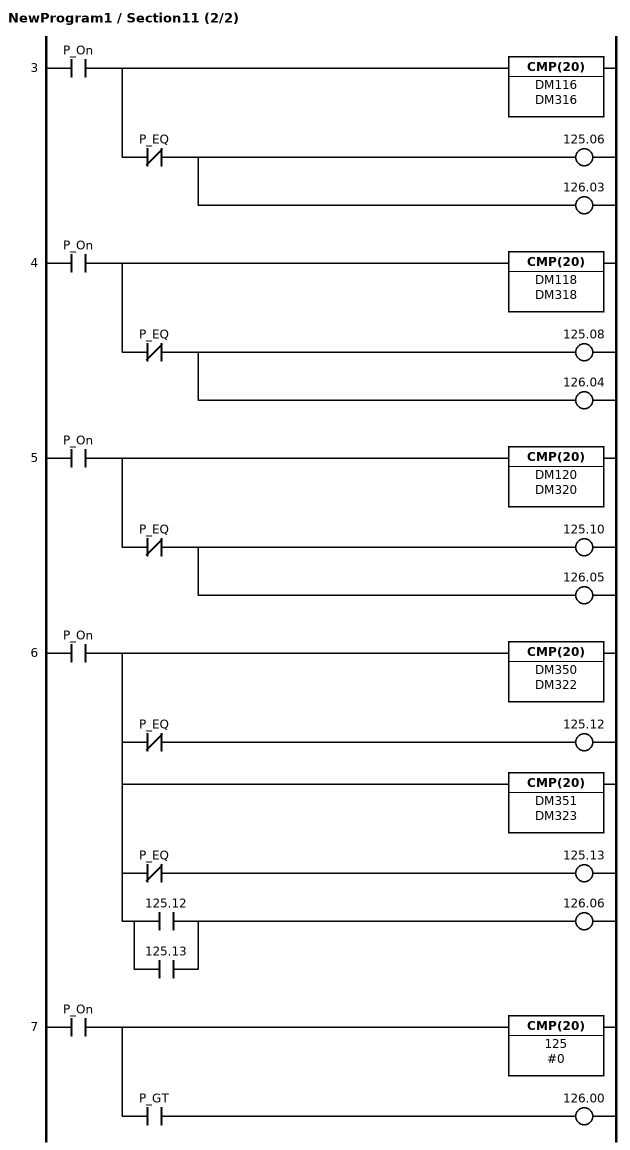
; [picture p48: NewProgram1 / Section11, rungs 3-7]
; rung 3
LD P_On
CMP(20) DM116 DM316
ANDNOT P_EQ
OUT 125.06
OUT 126.03
; rung 4
LD P_On
CMP(20) DM118 DM318
ANDNOT P_EQ
OUT 125.08
OUT 126.04
; rung 5
LD P_On
CMP(20) DM120 DM320
ANDNOT P_EQ
OUT 125.10
OUT 126.05
; rung 6
LD P_On
OUT TR0
CMP(20) DM350 DM322
ANDNOT P_EQ
OUT 125.12
LD TR0
CMP(20) DM351 DM323
ANDNOT P_EQ
OUT 125.13
LD TR0
LD 125.12
OR 125.13
ANDLD
OUT 126.06
; rung 7
LD P_On
CMP(20) 125 #0
AND P_GT
OUT 126.00

### Section Section12

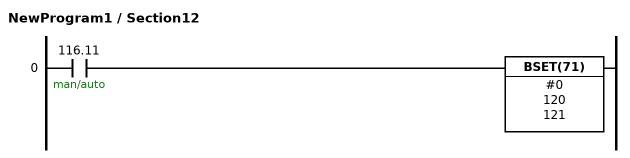
; rung 0
LD 116.11  ; man/auto
BSET(71) #0 120 121

### Section Section13

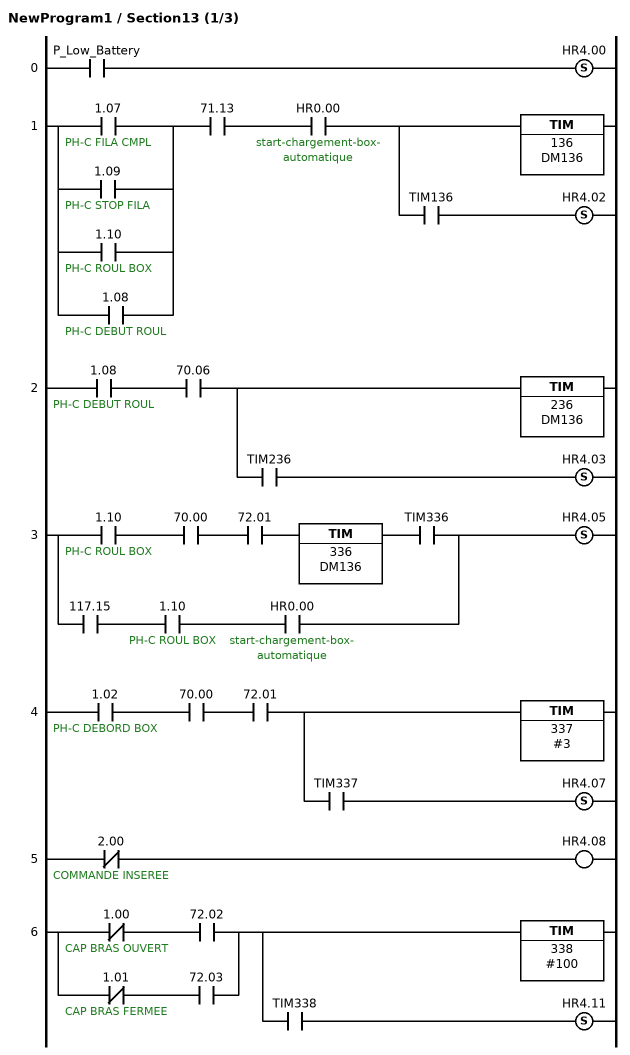
; rung 0
LD P_Low_Battery
SET HR4.00
; rung 1
LD 1.07  ; PH-C FILA CMPL
OR 1.09  ; PH-C STOP FILA
OR 1.10  ; PH-C ROUL BOX
OR 1.08  ; PH-C DEBUT ROUL
AND 71.13
AND HR0.00  ; start-chargement-box-automatique
TIM 136 DM136
AND TIM136
SET HR4.02
; rung 2
LD 1.08  ; PH-C DEBUT ROUL
AND 70.06
TIM 236 DM136
AND TIM236
SET HR4.03
; rung 3
LD 1.10  ; PH-C ROUL BOX
AND 70.00
AND 72.01
TIM 336 DM136
AND TIM336
LD 117.15
AND 1.10  ; PH-C ROUL BOX
AND HR0.00  ; start-chargement-box-automatique
ORLD
SET HR4.05
; rung 4
LD 1.02  ; PH-C DEBORD BOX
AND 70.00
AND 72.01
TIM 337 #3
AND TIM337
SET HR4.07
; rung 5
LDNOT 2.00  ; COMMANDE INSEREE
OUT HR4.08
; rung 6
LDNOT 1.00  ; CAP BRAS OUVERT
AND 72.02
LDNOT 1.01  ; CAP BRAS FERMEE
AND 72.03
ORLD
TIM 338 #100
AND TIM338
SET HR4.11

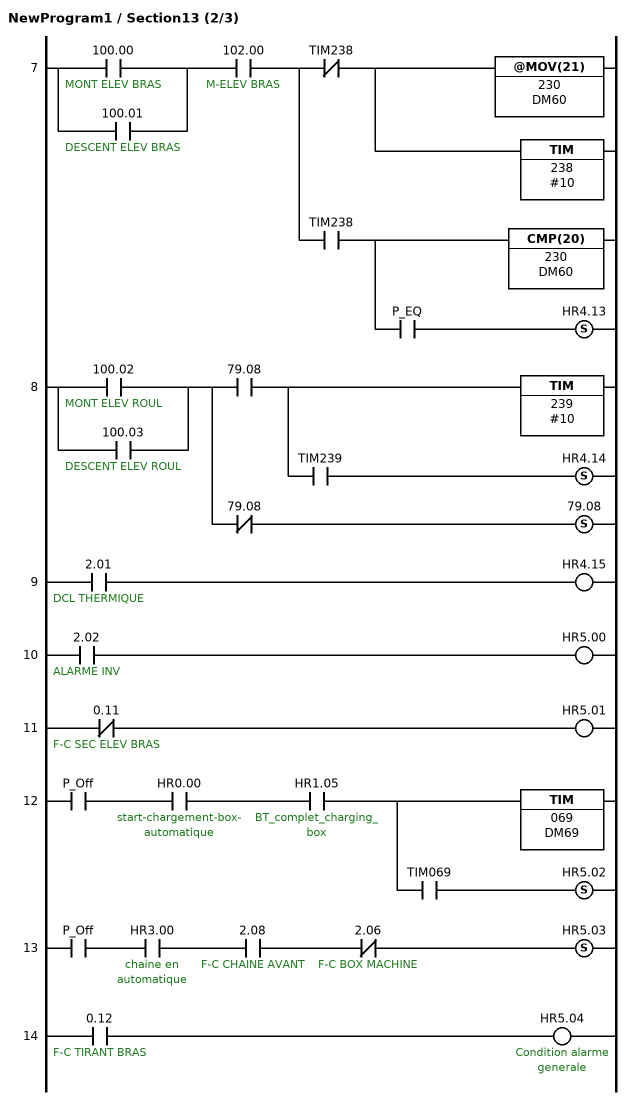
; rung 7
LD 100.00  ; MONT ELEV BRAS
OR 100.01  ; DESCENT ELEV BRAS
AND 102.00  ; M-ELEV BRAS
OUT TR0
ANDNOT TIM238
@MOV(21) 230 DM60
TIM 238 #10
LD TR0
AND TIM238
CMP(20) 230 DM60
AND P_EQ
SET HR4.13
; rung 8
LD 100.02  ; MONT ELEV ROUL
OR 100.03  ; DESCENT ELEV ROUL
OUT TR0
AND 79.08
TIM 239 #10
AND TIM239
SET HR4.14
LD TR0
ANDNOT 79.08
SET 79.08
; rung 9
LD 2.01  ; DCL THERMIQUE
OUT HR4.15
; rung 10
LD 2.02  ; ALARME INV
OUT HR5.00
; rung 11
LDNOT 0.11  ; F-C SEC ELEV BRAS
OUT HR5.01
; rung 12
LD P_Off
AND HR0.00  ; start-chargement-box-automatique
AND HR1.05  ; BT_complet_charging_box
TIM 069 DM69
AND TIM069
SET HR5.02
; rung 13
LD P_Off
AND HR3.00  ; chaine en automatique
AND 2.08  ; F-C CHAINE AVANT
ANDNOT 2.06  ; F-C BOX MACHINE
SET HR5.03
; rung 14
LD 0.12  ; F-C TIRANT BRAS
OUT HR5.04  ; Condition alarme generale

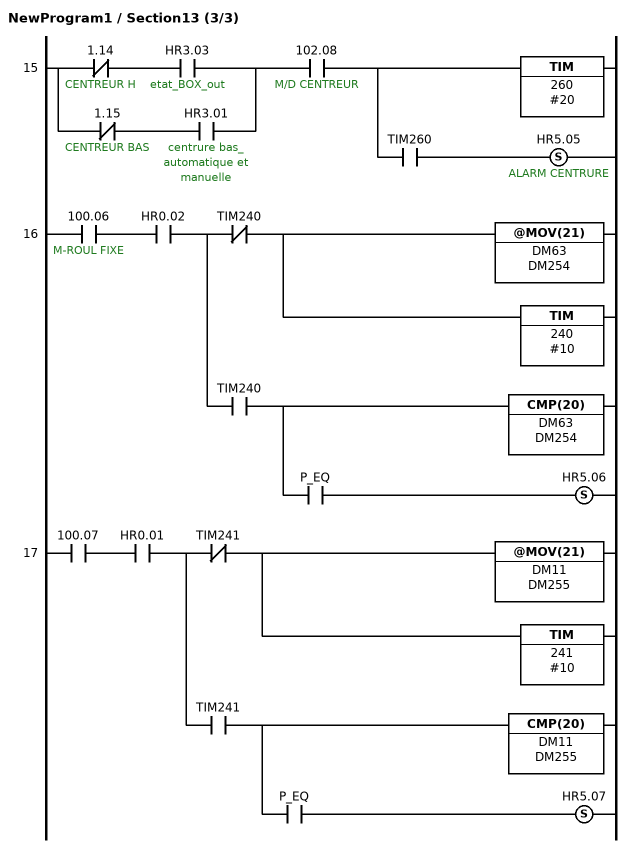
; rung 15
LDNOT 1.14  ; CENTREUR H
AND HR3.03  ; etat_BOX_out
LDNOT 1.15  ; CENTREUR BAS
AND HR3.01  ; centrure bas_automatique et manuelle
ORLD
AND 102.08  ; M/D CENTREUR
TIM 260 #20
AND TIM260
SET HR5.05  ; ALARM CENTRURE
; rung 16
LD 100.06  ; M-ROUL FIXE
AND HR0.02
OUT TR0
ANDNOT TIM240
@MOV(21) DM63 DM254
TIM 240 #10
LD TR0
AND TIM240
CMP(20) DM63 DM254
AND P_EQ
SET HR5.06
; rung 17
LD 100.07
AND HR0.01
OUT TR0
ANDNOT TIM241
@MOV(21) DM11 DM255
TIM 241 #10
LD TR0
AND TIM241
CMP(20) DM11 DM255
AND P_EQ
SET HR5.07

### Section consentement

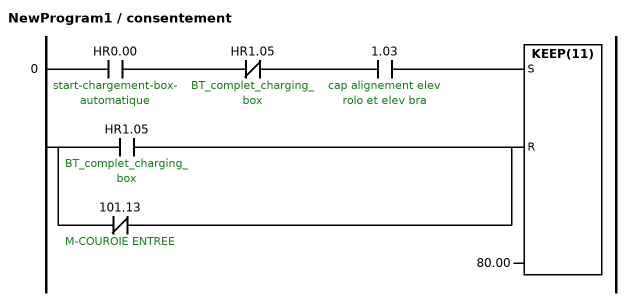
; rung 0
LD HR0.00  ; start-chargement-box-automatique
ANDNOT HR1.05  ; BT_complet_charging_box
AND 1.03  ; cap alignement elev rolo et elev bra
LD HR1.05  ; BT_complet_charging_box
ORNOT 101.13  ; M-COUROIE ENTREE
KEEP(11) 80.00

### Section Section15

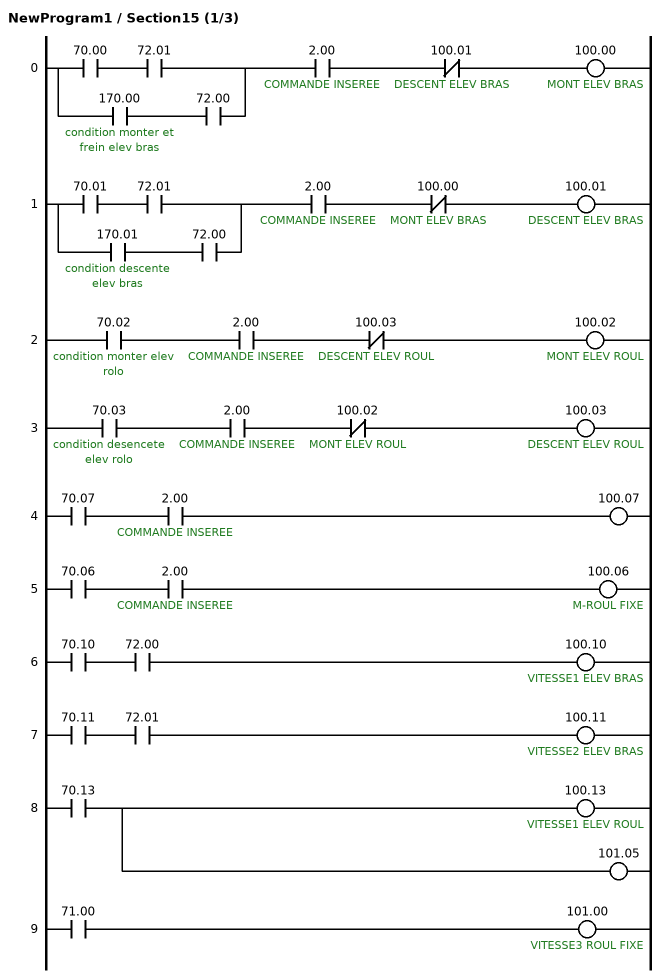
; rung 0
LD 70.00
AND 72.01
LD 170.00  ; condition monter et frein elev bras
AND 72.00
ORLD
AND 2.00  ; COMMANDE INSEREE
ANDNOT 100.01  ; DESCENT ELEV BRAS
OUT 100.00  ; MONT ELEV BRAS
; rung 1
LD 70.01
AND 72.01
LD 170.01  ; condition descente elev bras
AND 72.00
ORLD
AND 2.00  ; COMMANDE INSEREE
ANDNOT 100.00  ; MONT ELEV BRAS
OUT 100.01  ; DESCENT ELEV BRAS
; rung 2
LD 70.02  ; condition monter elev rolo
AND 2.00  ; COMMANDE INSEREE
ANDNOT 100.03  ; DESCENT ELEV ROUL
OUT 100.02  ; MONT ELEV ROUL
; rung 3
LD 70.03  ; condition desencete elev rolo
AND 2.00  ; COMMANDE INSEREE
ANDNOT 100.02  ; MONT ELEV ROUL
OUT 100.03  ; DESCENT ELEV ROUL
; rung 4
LD 70.07
AND 2.00  ; COMMANDE INSEREE
OUT 100.07
; rung 5
LD 70.06
AND 2.00  ; COMMANDE INSEREE
OUT 100.06  ; M-ROUL FIXE
; rung 6
LD 70.10
AND 72.00
OUT 100.10  ; VITESSE1 ELEV BRAS
; rung 7
LD 70.11
AND 72.01
OUT 100.11  ; VITESSE2 ELEV BRAS
; rung 8
LD 70.13
OUT 100.13  ; VITESSE1 ELEV ROUL
OUT 101.05
; rung 9
LD 71.00
OUT 101.00  ; VITESSE3 ROUL FIXE

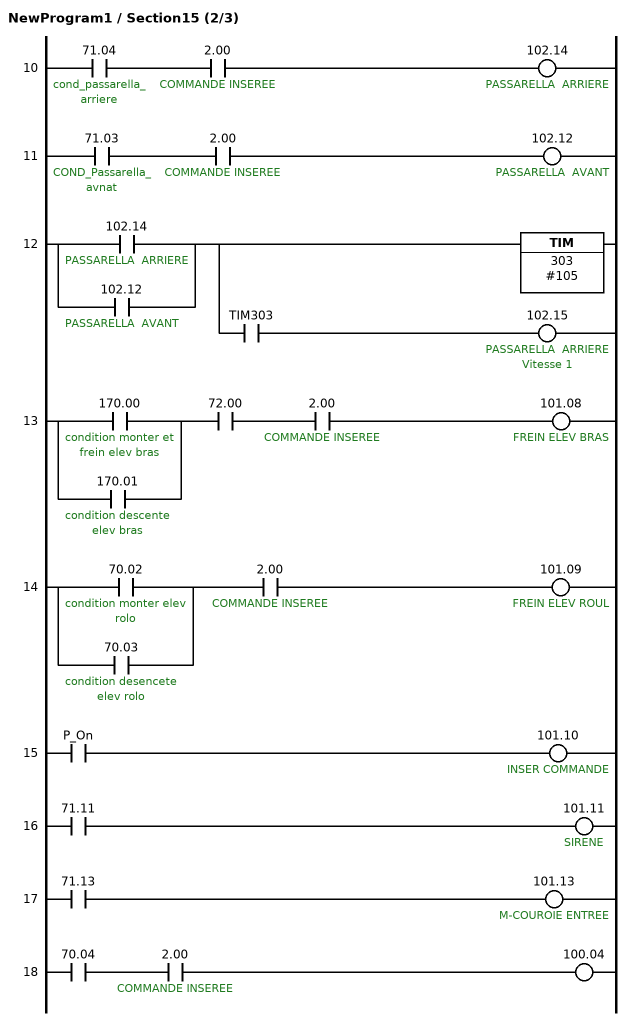
; rung 10
LD 71.04  ; cond_passarella_arriere
AND 2.00  ; COMMANDE INSEREE
OUT 102.14  ; PASSARELLA  ARRIERE
; rung 11
LD 71.03  ; COND_Passarella_avnat
AND 2.00  ; COMMANDE INSEREE
OUT 102.12  ; PASSARELLA  AVANT
; rung 12
LD 102.14  ; PASSARELLA  ARRIERE
OR 102.12  ; PASSARELLA  AVANT
TIM 303 #105
AND TIM303
OUT 102.15  ; PASSARELLA  ARRIERE Vitesse 1
; rung 13
LD 170.00  ; condition monter et frein elev bras
OR 170.01  ; condition descente elev bras
AND 72.00
AND 2.00  ; COMMANDE INSEREE
OUT 101.08  ; FREIN ELEV BRAS
; rung 14
LD 70.02  ; condition monter elev rolo
OR 70.03  ; condition desencete elev rolo
AND 2.00  ; COMMANDE INSEREE
OUT 101.09  ; FREIN ELEV ROUL
; rung 15
LD P_On
OUT 101.10  ; INSER COMMANDE
; rung 16
LD 71.11
OUT 101.11  ; SIRENE
; rung 17
LD 71.13
OUT 101.13  ; M-COUROIE ENTREE
; rung 18
LD 70.04
AND 2.00  ; COMMANDE INSEREE
OUT 100.04

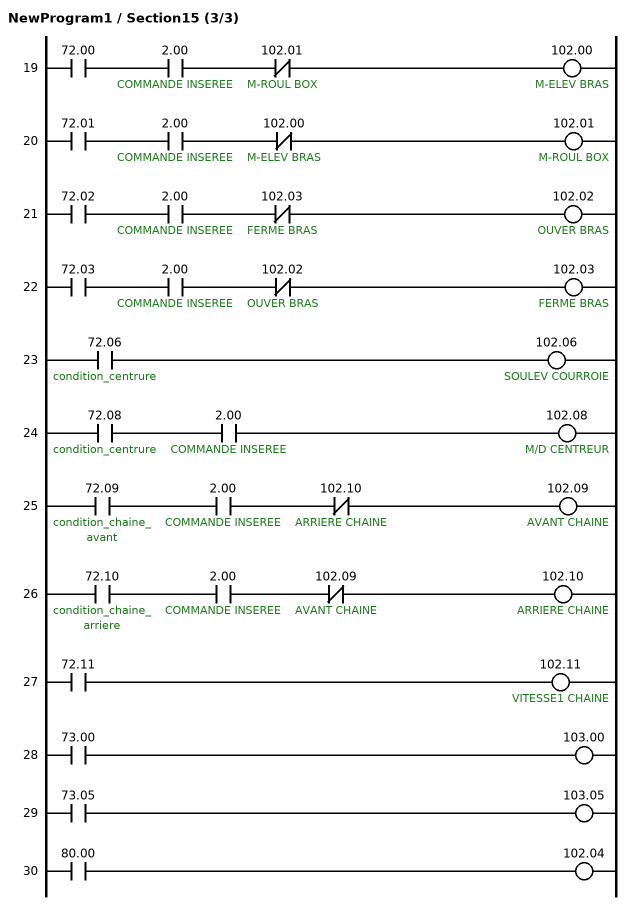
; rung 19
LD 72.00
AND 2.00  ; COMMANDE INSEREE
ANDNOT 102.01  ; M-ROUL BOX
OUT 102.00  ; M-ELEV BRAS
; rung 20
LD 72.01
AND 2.00  ; COMMANDE INSEREE
ANDNOT 102.00  ; M-ELEV BRAS
OUT 102.01  ; M-ROUL BOX
; rung 21
LD 72.02
AND 2.00  ; COMMANDE INSEREE
ANDNOT 102.03  ; FERME BRAS
OUT 102.02  ; OUVER BRAS
; rung 22
LD 72.03
AND 2.00  ; COMMANDE INSEREE
ANDNOT 102.02  ; OUVER BRAS
OUT 102.03  ; FERME BRAS
; rung 23
LD 72.06  ; condition_centrure
OUT 102.06  ; SOULEV COURROIE
; rung 24
LD 72.08  ; condition_centrure
AND 2.00  ; COMMANDE INSEREE
OUT 102.08  ; M/D CENTREUR
; rung 25
LD 72.09  ; condition_chaine_avant
AND 2.00  ; COMMANDE INSEREE
ANDNOT 102.10  ; ARRIERE CHAINE
OUT 102.09  ; AVANT CHAINE
; rung 26
LD 72.10  ; condition_chaine_arriere
AND 2.00  ; COMMANDE INSEREE
ANDNOT 102.09  ; AVANT CHAINE
OUT 102.10  ; ARRIERE CHAINE
; rung 27
LD 72.11
OUT 102.11  ; VITESSE1 CHAINE
; rung 28
LD 73.00
OUT 103.00
; rung 29
LD 73.05
OUT 103.05
; rung 30
LD 80.00
OUT 102.04

### Section Section16

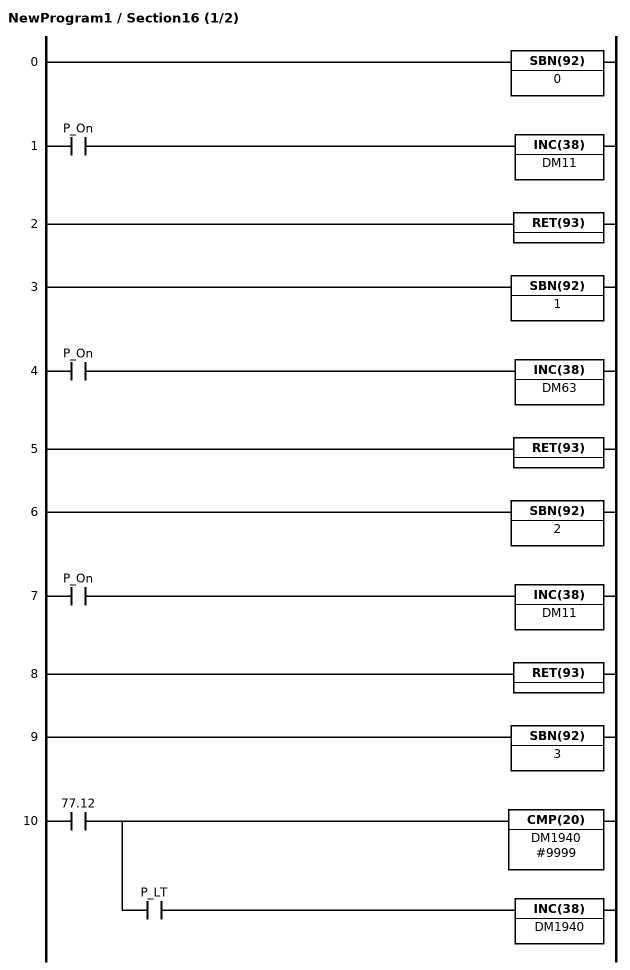
; rung 0
SBN(92) 0
; rung 1
LD P_On
INC(38) DM11
; rung 2
RET(93)
; rung 3
SBN(92) 1
; rung 4
LD P_On
INC(38) DM63
; rung 5
RET(93)
; rung 6
SBN(92) 2
; rung 7
LD P_On
INC(38) DM11
; rung 8
RET(93)
; rung 9
SBN(92) 3
; rung 10
LD 77.12
CMP(20) DM1940 #9999
AND P_LT
INC(38) DM1940

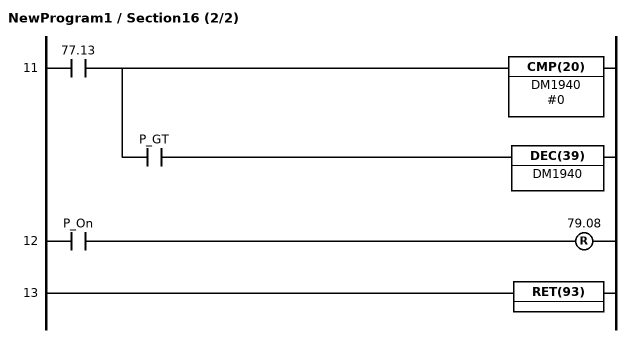
; rung 11
LD 77.13
CMP(20) DM1940 #0
AND P_GT
DEC(39) DM1940
; rung 12
LD P_On
RSET 79.08
; rung 13
RET(93)

### Section Section17
; rung 0
END(01)